// TIA Portal V19 export
FUNCTION "MatCounter_UPD" : Void   // FC103, LAD
TITLE = Update
// stored: Access Published, SetENOAutomatically false
   VAR_IN_OUT
      Data : "MatCountData";
   END_VAR
   VAR_TEMP
      AxDifference : LReal;
      HalfModule : LReal;
      HalfNegativeModule : LReal;
      AxFAKModule : LReal;
   END_VAR
BEGIN

REGION Network 1: AX FAK Module
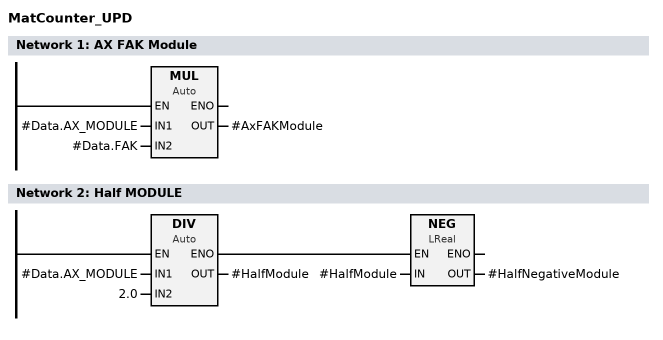
   RUNG wire#powerrail
      Mul(in1 := #Data.AX_MODULE, in2 := #Data.FAK, out => #AxFAKModule)
   END_RUNG
   // the same network as SCL:
   #AxFAKModule := #Data.AX_MODULE * #Data.FAK;
END_REGION

REGION Network 2: Half MODULE
   RUNG wire#powerrail
      Div(in1 := #Data.AX_MODULE, in2 := 2.0, out => #HalfModule)
      { S7_Templates := "SrcType := LReal" } Neg(in := #HalfModule, out => #HalfNegativeModule)
   END_RUNG
   // the same network as SCL:
   #HalfModule := #Data.AX_MODULE / 2.0;
   #HalfNegativeModule := -#HalfModule;
END_REGION

REGION Network 3 (SCL): Ax difference
   //=====================================================
   // CONTROLLO GIRO COMPLETO CONTEGGIO ASSE 
   //=====================================================
   #AxDifference := #Data.AxPosition - #Data.AxPositionPrevious;
   #Data.AxPositionPrevious := #Data.AxPosition;

   IF #AxDifference > #HalfModule THEN
       #Data.CounterOffset := #Data.CounterOffset - #AxFAKModule;
   ELSIF #AxDifference < #HalfNegativeModule THEN
       #Data.CounterOffset := #Data.CounterOffset + #AxFAKModule;
   END_IF;

   //=====================================================
   // COUNTER
   //=====================================================
   #Data.CounterValue := (#Data.AxPosition * #Data.FAK) + #Data.CounterOffset;

   IF #Data.CounterValue >= #Data.COUNTER_MODULE THEN
       #Data.CounterOffset := #Data.CounterOffset - #Data.COUNTER_MODULE;
       #Data.CounterValue := (#Data.AxPosition * #Data.FAK) + #Data.CounterOffset;

   ELSIF #Data.CounterValue < 0.0 THEN
       #Data.CounterOffset := #Data.CounterOffset + #Data.COUNTER_MODULE;
       #Data.CounterValue := (#Data.AxPosition * #Data.FAK) + #Data.CounterOffset;
   END_IF;


   IF ABS_LREAL(#Data.CounterValue - #Data.COUNTER_MODULE) < 0.01 THEN
       #Data.CounterValue := 0.0;
   END_IF;
END_REGION
END_FUNCTION
